// TIA Portal V20 export
DATA_BLOCK "Data"   // DB40
// stored: Access Published, MemoryReserve 100, Namespace Global
   VAR
      general : "LAF_typeGeneralStatus";   // Global status information
      unit : Array[0.._.NO_OF_UNITS] of "LAF_typeUnitInterface";   // Global information of units
   END_VAR
BEGIN
   // general.enablePower : Power is off. Switch on!
   unit[0].enableControlInterfaces.local := true;
   unit[0].enableControlInterfaces.hmi := False;
END_DATA_BLOCK
